INTERFACE ContinuousDrive

METHOD moveContinuous : BOOL
VAR_INPUT
	direction : MC_Direction;
END_VAR
END_METHOD

END_INTERFACE

(* stored: Version 1.1.0.1, ProductVersion 3.1.4024.11
   Itf ContinuousDrive: Id {27e7ee41-ea84-43ba-bbab-fcee94cc798c}
   Method moveContinuous: Id {aab498f2-15fd-447c-8469-faaeaeb26562} *)
